TYPE ST_Version :
STRUCT
	nMajor    		: DINT;
	nMinor    		: DINT;
	nBuild 			: DINT;
	nRevision 		: DINT;
	sVersion		: STRING;
END_STRUCT
END_TYPE

(* stored: Version 1.1.0.1, ProductVersion 3.1.4020.12
   DUT ST_Version: Id {d95edd5c-f829-4fd8-9a73-3d48dc09e0f6} *)
